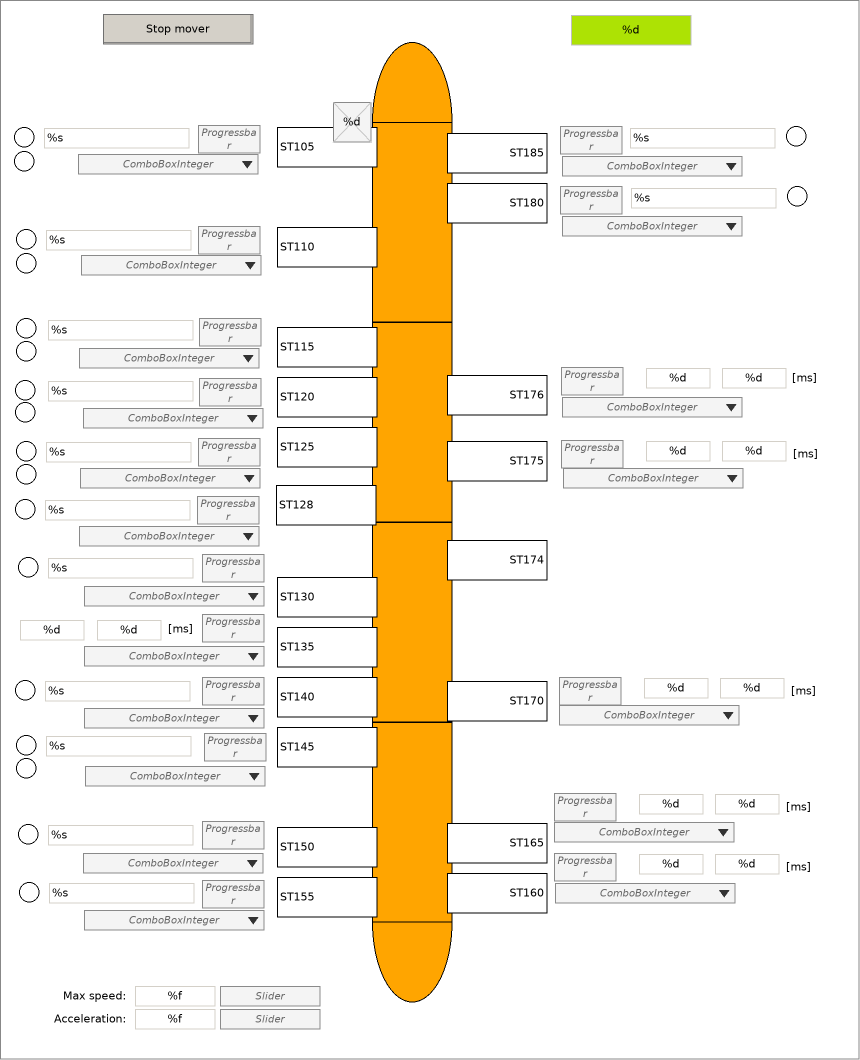
VISUALIZATION VISU_MoverView  // 860x1060
    Ellipse (372,842 80x160)
    Rectangle (372,722 80x200)
    Rectangle (372,522 80x200)
    Rectangle (372,322 80x200)
    Ellipse (372,42 80x160)
    Rectangle (372,122 80x200)
    Rectangle (447,183 100x40), "ST180", colour toggle: NOT GVL.st180_aut.xMoverPathFree
    Rectangle (447,375 100x40), "ST176", colour toggle: NOT GVL.st176_aut.xMoverPathFree
    Rectangle (447,441 100x40), "ST175", colour toggle: NOT GVL.st175_aut.xMoverPathFree
    Rectangle (447,681 100x40), "ST170", colour toggle: NOT GVL.st170_aut.xMoverPathFree
    Rectangle (447,823 100x40), "ST165", colour toggle: NOT GVL.st165_aut.xMoverPathFree
    Rectangle (447,873 100x40), "ST160", colour toggle: NOT GVL.st160_aut.xMoverPathFree
    Rectangle (277,877 100x40), "ST155", colour toggle: NOT GVL.st155_aut.xMoverPathFree
    Rectangle (447,133 100x40), "ST185", colour toggle: NOT GVL.st185_aut.xMoverPathFree
    Progressbar (560,186 62x28), variable: SIMU.iCompletionHMI[18]
    Progressbar (561,367 62x28), variable: SIMU.iCompletionHMI[17]
    Progressbar (561,440 62x28), variable: SIMU.iCompletionHMI[16]
    Progressbar (559,677 62x28), variable: SIMU.iCompletionHMI[14]
    Progressbar (554,793 62x28), variable: SIMU.iCompletionHMI[13]
    Progressbar (554,853 62x28), variable: SIMU.iCompletionHMI[12]
    Progressbar (202,880 62x28), variable: SIMU.iCompletionHMI[11]
    Progressbar (560,126 62x28), variable: SIMU.iCompletionHMI[19]
    Textfield (722,368 64x20), "%d", text variable: PERS.iStationTimeDef2[17]
        OnMouseDown: write the text variable via Default
    Label (777,363 55x30), "[ms]"
    Textfield (722,441 64x20), "%d", text variable: PERS.iStationTimeDef2[16]
        OnMouseDown: write the text variable via Default
    Label (778,439 55x30), "[ms]"
    Textfield (720,678 64x20), "%d", text variable: PERS.iStationTimeDef2[14]
        OnMouseDown: write the text variable via Default
    Label (776,676 55x30), "[ms]"
    Textfield (715,794 64x20), "%d", text variable: PERS.iStationTimeDef2[13]
        OnMouseDown: write the text variable via Default
    Label (771,792 55x30), "[ms]"
    Textfield (715,854 64x20), "%d", text variable: PERS.iStationTimeDef2[12]
        OnMouseDown: write the text variable via Default
    Label (771,852 55x30), "[ms]"
    Textfield (571,15 120x30), "%d", text variable: MAIN.MoverMan.PH_num, colour toggle: MAIN.MoverMan.PH_num>2
        OnMouseDown: write the text variable via Default
    ComboBoxInteger (562,156 180x20), variable: MAIN.MoverMan._StationList[18]._ApproachScenario
    ComboBoxInteger (562,216 180x20), variable: MAIN.MoverMan._StationList[17]._ApproachScenario
    ComboBoxInteger (562,397 180x20), variable: MAIN.MoverMan._StationList[16]._ApproachScenario
    ComboBoxInteger (563,468 180x20), variable: MAIN.MoverMan._StationList[16]._ApproachScenario
    ComboBoxInteger (559,705 180x20), variable: MAIN.MoverMan._StationList[14]._ApproachScenario
    ComboBoxInteger (554,822 180x20), variable: MAIN.MoverMan._StationList[13]._ApproachScenario
    ComboBoxInteger (555,883 180x20), variable: MAIN.MoverMan._StationList[12]._ApproachScenario
    ComboBoxInteger (84,910 180x20), variable: MAIN.MoverMan._StationList[11]._ApproachScenario
    Rectangle (277,827 100x40), "ST150", colour toggle: NOT GVL.st150_aut.xMoverPathFree
    Progressbar (202,821 62x28), variable: SIMU.iCompletionHMI[10]
    ComboBoxInteger (83,853 180x20), variable: MAIN.MoverMan._StationList[10]._ApproachScenario
    Rectangle (277,727 100x40), "ST145", colour toggle: NOT GVL.st145_aut.xMoverPathFree
    Progressbar (204,733 62x28), variable: SIMU.iCompletionHMI[9]
    ComboBoxInteger (85,766 180x20), variable: MAIN.MoverMan._StationList[9]._ApproachScenario
    Rectangle (277,677 100x40), "ST140", colour toggle: NOT GVL.st140_aut.xMoverPathFree
    Progressbar (202,677 62x28), variable: SIMU.iCompletionHMI[8]
    ComboBoxInteger (84,708 180x20), variable: MAIN.MoverMan._StationList[8]._ApproachScenario
    Textfield (97,620 64x20), "%d", text variable: PERS.iStationTimeDef2[7]
        OnMouseDown: write the text variable via Default
    Label (153,614 55x30), "[ms]"
    Rectangle (277,627 100x40), "ST135", colour toggle: NOT GVL.st135_aut.xMoverPathFree
    Progressbar (202,614 62x28), variable: SIMU.iCompletionHMI[7]
    ComboBoxInteger (84,646 180x20), variable: MAIN.MoverMan._StationList[7]._ApproachScenario
    Rectangle (277,577 100x40), "ST130", colour toggle: NOT GVL.st130_aut.xMoverPathFree
    Progressbar (202,554 62x28), variable: SIMU.iCompletionHMI[6]
    ComboBoxInteger (84,586 180x20), variable: MAIN.MoverMan._StationList[6]._ApproachScenario
    Rectangle (277,427 100x40), "ST125", colour toggle: NOT GVL.st125_aut.xMoverPathFree
    Progressbar (198,438 62x28), variable: SIMU.iCompletionHMI[5]
    ComboBoxInteger (80,468 180x20), variable: MAIN.MoverMan._StationList[5]._ApproachScenario
    Rectangle (277,377 100x40), "ST120", colour toggle: NOT GVL.st120_aut.xMoverPathFree
    Progressbar (199,378 62x28), variable: SIMU.iCompletionHMI[4]
    ComboBoxInteger (83,408 180x20), variable: MAIN.MoverMan._StationList[4]._ApproachScenario
    Rectangle (277,327 100x40), "ST115", colour toggle: NOT GVL.st115_aut.xMoverPathFree
    Progressbar (199,318 62x28), variable: SIMU.iCompletionHMI[3]
    ComboBoxInteger (79,348 180x20), variable: MAIN.MoverMan._StationList[3]._ApproachScenario
    Rectangle (277,227 100x40), "ST110", colour toggle: NOT GVL.st110_aut.xMoverPathFree
    Progressbar (198,226 62x28), variable: SIMU.iCompletionHMI[2]
    ComboBoxInteger (81,255 180x20), variable: MAIN.MoverMan._StationList[2]._ApproachScenario
    Rectangle (277,127 100x40), "ST105", colour toggle: NOT GVL.st105_aut.xMoverPathFree
    Progressbar (198,125 62x28), variable: SIMU.iCompletionHMI[1]
    ComboBoxInteger (78,154 180x20), variable: MAIN.MoverMan._StationList[1]._ApproachScenario
    Button (103,14 150x30), "Stop mover", colour toggle: MAIN.MoverMan.HMI_xStopMover
        toggle MAIN.MoverMan.HMI_xStopMover
    Textfield (135,986 80x20), "%f", text variable: SIMU.lrSpeedMover
    Textfield (135,1009 80x20), "%f", text variable: SIMU.lrAccelMover
    Label (29,986 100x20), "Max speed:"
    Label (29,1009 100x20), "Acceleration:"
    Slider (220,986 100x20), variable: SIMU.lrSpeedMover, scale 1..50
    Slider (220,1009 100x20), variable: SIMU.lrAccelMoverSlider, scale 0.1..1
    Textfield (20,620 64x20), "%d", text variable: PERS.iStationTimeDef1[7]
        OnMouseDown: write the text variable via Default
    Textfield (646,368 64x20), "%d", text variable: PERS.iStationTimeDef1[17]
        OnMouseDown: write the text variable via Default
    Textfield (646,441 64x20), "%d", text variable: PERS.iStationTimeDef1[16]
        OnMouseDown: write the text variable via Default
    Textfield (644,678 64x20), "%d", text variable: PERS.iStationTimeDef1[14]
        OnMouseDown: write the text variable via Default
    Textfield (639,794 64x20), "%d", text variable: PERS.iStationTimeDef1[13]
        OnMouseDown: write the text variable via Default
    Textfield (639,854 64x20), "%d", text variable: PERS.iStationTimeDef1[12]
        OnMouseDown: write the text variable via Default
    Textfield (46,230 145x20), "%s", text variable: GVL.st110_aut.fb_Pnp.sOUT_Step
    Textfield (48,320 145x20), "%s", text variable: GVL.st115_aut.fb_Pnp.sOUT_Step
    Textfield (48,381 145x20), "%s", text variable: GVL.st120_aut.fb_Pnp.sOUT_Step
    Rectangle (447,540 100x40), "ST174"
    Textfield (46,442 145x20), "%s", text variable: GVL.st125_aut.fb_Pnp.sOUT_Step
    Textfield (46,736 145x20), "%s", text variable: GVL.st145_aut.fb_Pnp.sOUT_Step
    Textfield (631,188 145x20), "%s", text variable: GVL.st180_aut.fb_Pnp.sOUT_Step
    Ellipse (16,229 20x20), colour toggle: GVL.st110_aut.xOUT_Ready
    Ellipse (16,318 20x20), colour toggle: GVL.st115_aut.xOUT_Ready
    Ellipse (15,380 20x20), colour toggle: GVL.st120_aut.xOUT_Ready
    Ellipse (16,441 20x20), colour toggle: GVL.st125_aut.xOUT_Ready
    Ellipse (16,735 20x20), colour toggle: GVL.st145_aut.xOUT_Ready
    Ellipse (787,186 20x20), colour toggle: GVL.st180_aut.xOUT_Ready
    Ellipse (16,253 20x20), colour toggle: GVL.st110_aut.fb_Feeder.xOUT_ErrFlag
    Ellipse (16,341 20x20), colour toggle: GVL.st115_aut.fb_Feeder.xOUT_ErrFlag
    Ellipse (15,402 20x20), colour toggle: GVL.st120_aut.fb_Feeder.xOUT_ErrFlag
    Ellipse (16,464 20x20), colour toggle: GVL.st125_aut.fb_Feeder.xOUT_ErrFlag
    Ellipse (16,758 20x20), colour toggle: GVL.st145_aut.fb_Feeder.xOUT_ErrFlag
    Textfield (630,128 145x20), "%s", text variable: GVL.st185_aut.fb_Pnp.sOUT_Step
    Ellipse (786,126 20x20), colour toggle: GVL.st185_aut.xOUT_Ready
    Textfield (48,558 145x20), "%s", text variable: GVL.st130_aut.fb_Dose.sOUT_Step
    Ellipse (18,557 20x20), colour toggle: GVL.st130_aut.xOUT_Ready
    Textfield (44,128 145x20), "%s", text variable: GVL.st105_aut.fb_Pnp.sOUT_Step
    Ellipse (14,127 20x20), colour toggle: GVL.st105_aut.xOUT_Ready
    Ellipse (14,151 20x20), colour toggle: GVL.st105_aut.fb_Feeder.xOUT_ErrFlag
    Textfield (45,681 145x20), "%s", text variable: GVL.st140_aut.fb_Measure.sOUT_Step
    Ellipse (15,680 20x20), colour toggle: GVL.st140_aut.xOUT_Ready
    Textfield (48,825 145x20), "%s", text variable: GVL.st150_aut.fb_Uss.sOUT_Step
    Ellipse (18,824 20x20), colour toggle: GVL.st150_aut.xOUT_Ready
    Textfield (49,883 145x20), "%s", text variable: GVL.st150_aut.fb_Uss.sOUT_Step
    Ellipse (19,882 20x20), colour toggle: GVL.st150_aut.xOUT_Ready
    Rectangle (276,485 100x40), "ST128", colour toggle: NOT GVL.st125_aut.xMoverPathFree
    Progressbar (197,496 62x28), variable: SIMU.iCompletionHMI[6]
    ComboBoxInteger (79,526 180x20), variable: MAIN.MoverMan._StationList[6]._ApproachScenario
    Textfield (45,500 145x20), "%s", text variable: GVL.st128_aut.fb_TubeCapCheck.sOUT_Step
    Ellipse (15,499 20x20), colour toggle: GVL.st128_aut.xOUT_Ready
    Image (333,102 38x40), "%d", text variable: MAIN.MoverMan._MoverList[1]._ID, colour toggle: MAIN.MoverMan._SimuMoverList[1]._xStuck, invisible if: MAIN.MoverMan._MoverList[1]._MoverAxis._iID>MAIN.MoverMan.MOVER_NUMBER, image: Custom.MoverSimu_final
        p3560616238: MAIN.MoverMan._MoverList[1]._MoverAxis.outSimuCurrentPos.x
        p2738717112: MAIN.MoverMan._MoverList[1]._MoverAxis.outSimuCurrentPos.y
        p2858320360: -MAIN.MoverMan._MoverList[1]._MoverAxis.outSimuCurrentRot
    Image (333,102 38x40), "%d", text variable: MAIN.MoverMan._MoverList[2]._ID, colour toggle: MAIN.MoverMan._SimuMoverList[2]._xStuck, invisible if: MAIN.MoverMan._MoverList[2]._MoverAxis._iID>MAIN.MoverMan.MOVER_NUMBER, image: Custom.MoverSimu_final
        p3560616238: MAIN.MoverMan._MoverList[2]._MoverAxis.outSimuCurrentPos.x
        p2738717112: MAIN.MoverMan._MoverList[2]._MoverAxis.outSimuCurrentPos.y
        p2858320360: -MAIN.MoverMan._MoverList[2]._MoverAxis.outSimuCurrentRot
    Image (333,102 38x40), "%d", text variable: MAIN.MoverMan._MoverList[3]._ID, colour toggle: MAIN.MoverMan._SimuMoverList[3]._xStuck, invisible if: MAIN.MoverMan._MoverList[3]._MoverAxis._iID>MAIN.MoverMan.MOVER_NUMBER, image: Custom.MoverSimu_final
        p3560616238: MAIN.MoverMan._MoverList[3]._MoverAxis.outSimuCurrentPos.x
        p2738717112: MAIN.MoverMan._MoverList[3]._MoverAxis.outSimuCurrentPos.y
        p2858320360: -MAIN.MoverMan._MoverList[3]._MoverAxis.outSimuCurrentRot
    Image (333,102 38x40), "%d", text variable: MAIN.MoverMan._MoverList[4]._ID, colour toggle: MAIN.MoverMan._SimuMoverList[4]._xStuck, invisible if: MAIN.MoverMan._MoverList[4]._MoverAxis._iID>MAIN.MoverMan.MOVER_NUMBER, image: Custom.MoverSimu_final
        p3560616238: MAIN.MoverMan._MoverList[4]._MoverAxis.outSimuCurrentPos.x
        p2738717112: MAIN.MoverMan._MoverList[4]._MoverAxis.outSimuCurrentPos.y
        p2858320360: -MAIN.MoverMan._MoverList[4]._MoverAxis.outSimuCurrentRot
    Image (333,102 38x40), "%d", text variable: MAIN.MoverMan._MoverList[5]._ID, colour toggle: MAIN.MoverMan._SimuMoverList[5]._xStuck, invisible if: MAIN.MoverMan._MoverList[5]._MoverAxis._iID>MAIN.MoverMan.MOVER_NUMBER, image: Custom.MoverSimu_final
        p3560616238: MAIN.MoverMan._MoverList[5]._MoverAxis.outSimuCurrentPos.x
        p2738717112: MAIN.MoverMan._MoverList[5]._MoverAxis.outSimuCurrentPos.y
        p2858320360: -MAIN.MoverMan._MoverList[5]._MoverAxis.outSimuCurrentRot
    Image (333,102 38x40), "%d", text variable: MAIN.MoverMan._MoverList[6]._ID, colour toggle: MAIN.MoverMan._SimuMoverList[6]._xStuck, invisible if: MAIN.MoverMan._MoverList[6]._MoverAxis._iID>MAIN.MoverMan.MOVER_NUMBER, image: Custom.MoverSimu_final
        p3560616238: MAIN.MoverMan._MoverList[6]._MoverAxis.outSimuCurrentPos.x
        p2738717112: MAIN.MoverMan._MoverList[6]._MoverAxis.outSimuCurrentPos.y
        p2858320360: -MAIN.MoverMan._MoverList[6]._MoverAxis.outSimuCurrentRot
    Image (333,102 38x40), "%d", text variable: MAIN.MoverMan._MoverList[7]._ID, colour toggle: MAIN.MoverMan._SimuMoverList[7]._xStuck, invisible if: MAIN.MoverMan._MoverList[7]._MoverAxis._iID>MAIN.MoverMan.MOVER_NUMBER, image: Custom.MoverSimu_final
        p3560616238: MAIN.MoverMan._MoverList[7]._MoverAxis.outSimuCurrentPos.x
        p2738717112: MAIN.MoverMan._MoverList[7]._MoverAxis.outSimuCurrentPos.y
        p2858320360: -MAIN.MoverMan._MoverList[7]._MoverAxis.outSimuCurrentRot
    Image (333,102 38x40), "%d", text variable: MAIN.MoverMan._MoverList[8]._ID, colour toggle: MAIN.MoverMan._SimuMoverList[8]._xStuck, invisible if: MAIN.MoverMan._MoverList[8]._MoverAxis._iID>MAIN.MoverMan.MOVER_NUMBER, image: Custom.MoverSimu_final
        p3560616238: MAIN.MoverMan._MoverList[8]._MoverAxis.outSimuCurrentPos.x
        p2738717112: MAIN.MoverMan._MoverList[8]._MoverAxis.outSimuCurrentPos.y
        p2858320360: -MAIN.MoverMan._MoverList[8]._MoverAxis.outSimuCurrentRot
    Image (333,102 38x40), "%d", text variable: MAIN.MoverMan._MoverList[9]._ID, colour toggle: MAIN.MoverMan._SimuMoverList[9]._xStuck, invisible if: MAIN.MoverMan._MoverList[9]._MoverAxis._iID>MAIN.MoverMan.MOVER_NUMBER, image: Custom.MoverSimu_final
        p3560616238: MAIN.MoverMan._MoverList[9]._MoverAxis.outSimuCurrentPos.x
        p2738717112: MAIN.MoverMan._MoverList[9]._MoverAxis.outSimuCurrentPos.y
        p2858320360: -MAIN.MoverMan._MoverList[9]._MoverAxis.outSimuCurrentRot
    Image (333,102 38x40), "%d", text variable: MAIN.MoverMan._MoverList[10]._ID, colour toggle: MAIN.MoverMan._SimuMoverList[10]._xStuck, invisible if: MAIN.MoverMan._MoverList[10]._MoverAxis._iID>MAIN.MoverMan.MOVER_NUMBER, image: Custom.MoverSimu_final
        p3560616238: MAIN.MoverMan._MoverList[10]._MoverAxis.outSimuCurrentPos.x
        p2738717112: MAIN.MoverMan._MoverList[10]._MoverAxis.outSimuCurrentPos.y
        p2858320360: -MAIN.MoverMan._MoverList[10]._MoverAxis.outSimuCurrentRot
    Image (333,102 38x40), "%d", text variable: MAIN.MoverMan._MoverList[11]._ID, colour toggle: MAIN.MoverMan._SimuMoverList[11]._xStuck, invisible if: MAIN.MoverMan._MoverList[11]._MoverAxis._iID>MAIN.MoverMan.MOVER_NUMBER, image: Custom.MoverSimu_final
        p3560616238: MAIN.MoverMan._MoverList[11]._MoverAxis.outSimuCurrentPos.x
        p2738717112: MAIN.MoverMan._MoverList[11]._MoverAxis.outSimuCurrentPos.y
        p2858320360: -MAIN.MoverMan._MoverList[11]._MoverAxis.outSimuCurrentRot
    Image (333,102 38x40), "%d", text variable: MAIN.MoverMan._MoverList[12]._ID, colour toggle: MAIN.MoverMan._SimuMoverList[12]._xStuck, invisible if: MAIN.MoverMan._MoverList[12]._MoverAxis._iID>MAIN.MoverMan.MOVER_NUMBER, image: Custom.MoverSimu_final
        p3560616238: MAIN.MoverMan._MoverList[12]._MoverAxis.outSimuCurrentPos.x
        p2738717112: MAIN.MoverMan._MoverList[12]._MoverAxis.outSimuCurrentPos.y
        p2858320360: -MAIN.MoverMan._MoverList[12]._MoverAxis.outSimuCurrentRot
    Image (333,102 38x40), "%d", text variable: MAIN.MoverMan._MoverList[13]._ID, colour toggle: MAIN.MoverMan._SimuMoverList[13]._xStuck, invisible if: MAIN.MoverMan._MoverList[13]._MoverAxis._iID>MAIN.MoverMan.MOVER_NUMBER, image: Custom.MoverSimu_final
        p3560616238: MAIN.MoverMan._MoverList[13]._MoverAxis.outSimuCurrentPos.x
        p2738717112: MAIN.MoverMan._MoverList[13]._MoverAxis.outSimuCurrentPos.y
        p2858320360: -MAIN.MoverMan._MoverList[13]._MoverAxis.outSimuCurrentRot
    Image (333,102 38x40), "%d", text variable: MAIN.MoverMan._MoverList[14]._ID, colour toggle: MAIN.MoverMan._SimuMoverList[14]._xStuck, invisible if: MAIN.MoverMan._MoverList[14]._MoverAxis._iID>MAIN.MoverMan.MOVER_NUMBER, image: Custom.MoverSimu_final
        p3560616238: MAIN.MoverMan._MoverList[14]._MoverAxis.outSimuCurrentPos.x
        p2738717112: MAIN.MoverMan._MoverList[14]._MoverAxis.outSimuCurrentPos.y
        p2858320360: -MAIN.MoverMan._MoverList[14]._MoverAxis.outSimuCurrentRot
    Image (333,102 38x40), "%d", text variable: MAIN.MoverMan._MoverList[15]._ID, colour toggle: MAIN.MoverMan._SimuMoverList[15]._xStuck, invisible if: MAIN.MoverMan._MoverList[15]._MoverAxis._iID>MAIN.MoverMan.MOVER_NUMBER, image: Custom.MoverSimu_final
        p3560616238: MAIN.MoverMan._MoverList[15]._MoverAxis.outSimuCurrentPos.x
        p2738717112: MAIN.MoverMan._MoverList[15]._MoverAxis.outSimuCurrentPos.y
        p2858320360: -MAIN.MoverMan._MoverList[15]._MoverAxis.outSimuCurrentRot
    Image (333,102 38x40), "%d", text variable: MAIN.MoverMan._MoverList[16]._ID, colour toggle: MAIN.MoverMan._SimuMoverList[16]._xStuck, invisible if: MAIN.MoverMan._MoverList[16]._MoverAxis._iID>MAIN.MoverMan.MOVER_NUMBER, image: Custom.MoverSimu_final
        p3560616238: MAIN.MoverMan._MoverList[16]._MoverAxis.outSimuCurrentPos.x
        p2738717112: MAIN.MoverMan._MoverList[16]._MoverAxis.outSimuCurrentPos.y
        p2858320360: -MAIN.MoverMan._MoverList[16]._MoverAxis.outSimuCurrentRot
    Image (333,102 38x40), "%d", text variable: MAIN.MoverMan._MoverList[17]._ID, colour toggle: MAIN.MoverMan._SimuMoverList[17]._xStuck, invisible if: MAIN.MoverMan._MoverList[17]._MoverAxis._iID>MAIN.MoverMan.MOVER_NUMBER, image: Custom.MoverSimu_final
        p3560616238: MAIN.MoverMan._MoverList[17]._MoverAxis.outSimuCurrentPos.x
        p2738717112: MAIN.MoverMan._MoverList[17]._MoverAxis.outSimuCurrentPos.y
        p2858320360: -MAIN.MoverMan._MoverList[17]._MoverAxis.outSimuCurrentRot
    Image (333,102 38x40), "%d", text variable: MAIN.MoverMan._MoverList[18]._ID, colour toggle: MAIN.MoverMan._SimuMoverList[18]._xStuck, invisible if: MAIN.MoverMan._MoverList[18]._MoverAxis._iID>MAIN.MoverMan.MOVER_NUMBER, image: Custom.MoverSimu_final
        p3560616238: MAIN.MoverMan._MoverList[18]._MoverAxis.outSimuCurrentPos.x
        p2738717112: MAIN.MoverMan._MoverList[18]._MoverAxis.outSimuCurrentPos.y
        p2858320360: -MAIN.MoverMan._MoverList[18]._MoverAxis.outSimuCurrentRot
    Image (333,102 38x40), "%d", text variable: MAIN.MoverMan._MoverList[19]._ID, colour toggle: MAIN.MoverMan._SimuMoverList[19]._xStuck, invisible if: MAIN.MoverMan._MoverList[19]._MoverAxis._iID>MAIN.MoverMan.MOVER_NUMBER, image: Custom.MoverSimu_final
        p3560616238: MAIN.MoverMan._MoverList[19]._MoverAxis.outSimuCurrentPos.x
        p2738717112: MAIN.MoverMan._MoverList[19]._MoverAxis.outSimuCurrentPos.y
        p2858320360: -MAIN.MoverMan._MoverList[19]._MoverAxis.outSimuCurrentRot
END_VISUALIZATION

(* stored: Version 1.1.0.1, ProductVersion 3.1.4024.6
   Visu VISU_MoverView: Id {b2791c27-3f2c-4c3c-8103-f3f02d0db95f} *)
